FUNCTION_BLOCK FB_SafetyGen2  EXTENDS FB_Safety

VAR_INPUT
END_VAR

VAR_OUTPUT
	bVoltageSafe			: BOOL;
	bToolTempSafe			: BOOL;
	//eCurrentState			: E_SafetyState;
END_VAR

VAR
	
	bEmergencyStop			AT %I* : BOOL;	//Notaus ist gedrückt
	bInterlockIsLocked		AT %I* : BOOL;	//Interlock ist ordnungsgemäß verriegelt
	bBoxContactsClosed		AT %I* : BOOL;	//Sicherheitskontakte der Sicherheitsbox geschlossen
	bDriveIsSafe			AT %I* : BOOL;	//Sicherheitsrelais der Antriebe haben nicht angezogen
	bMesIsSafe				AT %I* : BOOL;	//Sicherheitsrelais in MES-Box hat nicht angezogen
	 
	nTwinSafeGrpState		AT %I* : USINT;
	
	bRequDriveOn			AT %Q* : BOOL;	//Request an TwinSafe Gruppe die Drives freizugeben (Relais einschalten)
	bRequMesOn				AT %Q* : BOOL;	//Request an TwinSafe Gruppe die MES freizugeben (Relais im HV-Generator einschalten)
	bRequUnlock				AT %Q* : BOOL;	//Request an TwinSafe Gruppe die Sicherheitsbox zu entriegeln

	bErrAckTwinSafeGrp		AT %Q* : BOOL;	//Error in TwinSafe Gruppe zurücksetzen
	
	nSubstate				: USINT := 0;
	nActionState			: USINT := 0;
	eStateRequest			: E_SafetyState;
	
	bResetError				: BOOL;
	bLock					: BOOL;
	bUnlock					: BOOL;
	bMonitor				: BOOL;
	nStateAction			: USINT;
	timer					: TON;
	i						: UINT;
	stPosition				: ST_3DPoint;
	
	stError					: ST_Error;
	stActionData			: ST_ActionData;
	
	pXYDrive				: POINTER TO FB_XYDriveBase;
	
END_VAR

VAR CONSTANT
	rSafePositionX			: REAL := 400000.0;
	rSafePositionY			: REAL := 200000.0;
	nSafeTemp				: UINT := 500; //50°C
END_VAR

CASE eCurrentState OF
	E_SafetyState.Init:
		//Dieser State wird nur am Anfang einmal durchlaufen und falls die TwinSafe Gruppe in Error ist,
		//wird dieser zurückgesetzt
		IF nSubState = 0 THEN
			IF nTwinSafeGrpState <> 1 THEN
				nSubState := 1;
			ELSE
				nSubState := 80;
			END_IF
		END_IF
		//Error zurücksetzen
		IF nSubState = 1 THEN
			A_ResetError();
			IF nStateAction >= 80 THEN
				IF nStateAction = 99 THEN
					nSubState := 99;
				ELSE
					nSubState := 80;
				END_IF
				nStateAction := 0;
			END_IF
		END_IF
		//weiterschalten
		IF nSubState >= 80 THEN
			IF nSubState = 99 THEN
				eCurrentState := E_SafetyState.Error;
			ELSE
				//folgende States sind von hier aus möglich
				//1: EmergencyStop wenn Notaustaster gedrückt
				//2: Locked wenn Interlock verriegelt (MES ist dabei egal)
				//3: UnlockedBoxCtcOpen wenn Interlock entriegelt und der Betätiger im Interlock oder ein anderer Sicherheitskontakt unterbrochen
				//4: UnlockedBoxCtcClosed wenn Interlock entriegelt und der Betätiger im Interlock und alle anderen Sicherheitskontakte geschlossen
				IF bEmergencyStop THEN
					eCurrentState := E_SafetyState.EmergencyStopPressed;
				ELSIF bInterlockIsLocked  THEN
					eCurrentState := E_SafetyState.Locked;
				ELSIF NOT bInterlockIsLocked AND NOT bBoxContactsClosed THEN
					eCurrentState := E_SafetyState.UnlockedBoxCtcOpen;
				ELSIF NOT bInterlockIsLocked AND bBoxContactsClosed THEN
					eCurrentState := E_SafetyState.UnlockedBoxCtcClosed;
				END_IF
			END_IF
			nSubState := 0;
		END_IF
	
	E_SafetyState.Locked:
		//folgende States sind von hier aus möglich
		//1: Error wenn: BoxContact geöffnet wird 
		//				 Interlock durch Schlüssel geöffnet wird ("bInterlockIsLocked" wechselt zu false)
		//				 SaftyLogic meldet Error
		//				 A_Unlock() mit State 99(Error) endet
		//2: EmergencyStop wenn Notaustaster gedrückt
		//3: UnlockedBoxCtcClosed wenn A_Unlock() State 80(Succes) endet
		bRequDriveOn := TRUE;
		IF nSubstate = 0 THEN //wartet auf StateRequest und überwacht
			IF NOT (bInterlockIsLocked AND bBoxContactsClosed AND nTwinSafeGrpState = 1) THEN //führt zu Error
				eCurrentState := E_SafetyState.Error;
			ELSIF bEmergencyStop THEN
				eCurrentState := E_SafetyState.EmergencyStopPressed;
			ELSIF eStateRequest = E_SafetyState.UnlockedBoxCtcClosed THEN
				nSubstate := 1;
			END_IF
		ELSIF nSubstate = 1 THEN //führt A_Unlock() aus
			A_Unlock();
			IF nStateAction >= 80 THEN
				IF nStateAction = 99 THEN
					eCurrentState := E_SafetyState.Error;
				ELSE
					eCurrentState := E_SafetyState.UnlockedBoxCtcClosed;
				END_IF
				nSubState := 0;
				nStateAction := 0;
			END_IF
		END_IF

		//Wenn dieser State verlassen wird, dann in jedem Fall bRequDriveOn und bRequMesOn zurücknehmen
		IF eCurrentState <> E_SafetyState.Locked THEN
			bRequDriveOn := FALSE;
			bRequMesOn := FALSE;
		END_IF
		
	E_SafetyState.UnlockedBoxCtcClosed:
		//folgende States sind von hier aus möglich
		//1: Error wenn: SaftyLogic meldet Error oder A_Locked() mit State 99 (Error) endet
		//2: EmergencyStop wenn Notaustaster gedrückt
		//3: UnlockedBoxCtcOpen wenn: BoxContact geöffnet wird 
		//							  Interlock durch Schlüssel geöffnet wird ("bInterlockIsLocked" wechselt zu false)
		//4: Locked wenn A_Lock() State 80(Succes) endet

		IF nSubstate = 0 THEN //wartet auf StateRequest und überwacht
			IF NOT (bInterlockIsLocked AND bBoxContactsClosed AND nTwinSafeGrpState = 1) THEN //führt zu Error
				eCurrentState := E_SafetyState.Error;
			ELSIF bEmergencyStop THEN
				eCurrentState := E_SafetyState.EmergencyStopPressed;
			ELSIF eStateRequest = E_SafetyState.Locked THEN
				nSubstate := 1;
			END_IF
		ELSIF nSubstate = 1 THEN //führt A_Lock() aus
			A_Lock();
			IF nStateAction >= 80 THEN
				IF nStateAction = 99 THEN
					eCurrentState := E_SafetyState.Error;
				ELSE
					eCurrentState := E_SafetyState.Locked;
				END_IF
				nSubState := 0;
				nStateAction := 0;
			END_IF
		END_IF
		
	E_SafetyState.UnlockedBoxCtcOpen:
		//folgende States sind von hier aus möglich
		//1: Error wenn: SaftyLogic meldet Error
		//2: EmergencyStop wenn Notaustaster gedrückt wird
		//3: UnlockedBoxCtcClosed wenn BoxContact geschlossen wird
		IF nTwinSafeGrpState <> 1 THEN
			eCurrentState := E_SafetyState.Error;
		ELSIF bEmergencyStop THEN
			eCurrentState := E_SafetyState.EmergencyStopPressed;
		ELSIF bBoxContactsClosed THEN
			eCurrentState := E_SafetyState.UnlockedBoxCtcClosed;
		END_IF
	
	E_SafetyState.EmergencyStopPressed:
		//folgende States sind von hier aus möglich
		//1: Error wenn: SaftyLogic meldet Error
		//2: EmergencyStopReleased wenn der Notaustaster wieder freigegeben wird
		IF nTwinSafeGrpState <> 1 THEN
			eCurrentState := E_SafetyState.Error;
		ELSIF NOT bEmergencyStop THEN
			eCurrentState := E_SafetyState.EmergencyStopReleased;
		END_IF
	E_SafetyState.EmergencyStopReleased:
		//folgende States sind von hier aus möglich
		//1: Error wenn: SaftyLogic meldet Error
		//2: in vorherigen State wechseln
END_CASE

ACTION A_Lock:

END_ACTION

ACTION A_ResetError:

END_ACTION

ACTION A_Unlock:

END_ACTION

METHOD M_LockUnlock : ERRORID
VAR_INPUT
	bLock : BOOL;
END_VAR
END_METHOD

METHOD M_ResetError
VAR_INPUT
END_VAR
bResetError := TRUE;
END_METHOD

PROPERTY P_nSafeToolTemp : UINT
GET
P_nSafeToolTemp := nSafeTemp;
END_GET
END_PROPERTY

PROPERTY P_rSafePositionX : REAL
GET
P_rSafePositionX := rSafePositionX;
END_GET
END_PROPERTY

PROPERTY P_rSafePositionY : REAL
GET
P_rSafePositionY := rSafePositionY;
END_GET
END_PROPERTY

END_FUNCTION_BLOCK

(* stored: Version 1.1.0.1, ProductVersion 3.1.4022.10
   POU FB_SafetyGen2: Id {81d7b58a-4596-42bc-80ea-8d35bfefe859}, SpecialFunc None
   Action A_Lock: Id {5bba04f3-9455-47c7-a3d9-f355086fe15f}
   Action A_ResetError: Id {7b8e6dbf-2fe5-4e43-90f8-80b6f4f5ad7f}
   Action A_Unlock: Id {814b23ae-ab9a-4f78-bfea-d6cf67671837}
   Method M_LockUnlock: Id {58aab17f-a3d7-4f3c-9c5b-0128e4fa3a9e}
   Method M_ResetError: Id {c0082624-8d33-42d2-80a1-7b00b769a716}
   Property P_nSafeToolTemp: Id {0f0c7e52-30a8-40d4-91a6-ce3b8f73b033}
   Get Get: Id {92004936-9027-499b-bdbf-96482aa6cda8}
   Property P_rSafePositionX: Id {8b4e1430-2219-429d-9392-fc171d48719d}
   Get Get: Id {1605b253-8c1a-47ff-b732-3135faf503a8}
   Property P_rSafePositionY: Id {a099f67b-8d96-4122-a37e-132c8b39ab3f}
   Get Get: Id {f8001ab2-f33b-40a0-8106-e33fda58c242} *)
